(* Logix 5000 project; controller cal1632 1756-L62 rev 16.20; software revision 16.05; part 53 of 57 *)
(* tags used below, declared in another part *)
   AFI : BOOL;
   FAULT : BOOL;
   p01_recipe_active : recipe;
   p01r02_plc_scan_time_in_sec : REAL;
   p01r09_pb_global_reset : BOOL;
   p01r09_request_line_jog : BOOL;
   p01r13_line_running : BOOL;
   p01r13_line_slow_ramp : BOOL;
   p01r13_permissive_drives : BOOL;
   p02_real_from_hmi : hmi_real;
   p25_ao_selected_speed : REAL;
   p25r09_mode_thread : BOOL;
   p25r09_pb_jog_fwd : BOOL;
   p25r09_pb_jog_rev : BOOL;
   p29_ai_wa_torque : REAL;
   p29_ai_wb_torque : REAL;
   p29_ai_wdr_lc : REAL;
   p29_ao_wdra_selected_speed : REAL;
   p29_ao_wdrb_selected_speed : REAL;
   p29_di_wa_brake : BOOL;
   p29_di_wa_motor : BOOL;
   p29_di_wdr_a_start : BOOL;
   p29_di_wdr_a_stop : BOOL;
   p29_di_wdr_b_start : BOOL;
   p29_di_wdr_b_stop : BOOL;
   p29_di_wdr_index_fwd : BOOL;
   p29_di_wdr_jog : BOOL;
   p29_param_soak : REAL;
   p29_param_winder_jog_speed : REAL;
   p29_wda_control_word : INT;
   p29_wda_status_word : INT;
   p29_wda_vfd : ABB_PROTOCOL_VFD;
   p29_wdb_control_word : INT;
   p29_wdb_status_word : INT;
   p29_wdb_vfd : ABB_PROTOCOL_VFD;
   p29r02_tension_dev_max : REAL;
   p29r02_tension_dev_min : REAL;
   p29r02_wa_calc_torque_ref : REAL;
   p29r02_wb_calc_torque_ref : REAL;
   p29r09_torque_mode : BOOL;
   p29r09_winder_a_active : BOOL;
   p29r09_winder_b_active : BOOL;
   p29r10_index_active : BOOL;
   p29r10_speed_offset : REAL;
   p29r11_index_active : BOOL;
   p29r11_speed_offset : REAL;
   p29r15 : routine;
   p29r15_accel_rate : REAL;
   p29r15_ao_torque : REAL;
   p29r15_const_torque_ref : REAL;
   p29r15_decel_rate : REAL;
   p29r15_fast_accel_rate : REAL;
   p29r15_fast_decel_rate : REAL;
   p29r15_index_start_torque : REAL;
   p29r15_jog_torque_ref : REAL;
   p29r15_request_jog_fwd : BOOL;
   p29r15_request_run : BOOL;
   p29r15_request_thread_fwd : BOOL;
   p29r15_request_thread_rev : BOOL;
   p29r15_run_permissive : BOOL;
   p29r15_selected_speed : REAL;
   p29r15_selected_torque : REAL;
   p29r15_soak_active : BOOL;
   p29r15_state : DINT;
   p29r15_tension_ok : BOOL;
   p29r15_thread_torque_ref : REAL;
   p29r15_timer_fault : TIMER[10];
   p29r15_timer_warning : TIMER[4];
   p29r15_torque_acc_rate : REAL;
   p29r15_torque_boost_acc_rate : REAL;
   p29r15_torque_boost_dec_rate : REAL;
   p29r15_torque_boost_ref : REAL;
   p29r15_torque_boost_timer : TIMER;
   p29r15_torque_dec_rate : REAL;
   p29r15_torque_fast_acc_rate : REAL;
   p29r15_torque_fast_dec_rate : REAL;
   p29r15_torque_high_ref : REAL;
   p29r15_torque_low_ref : REAL;
   p29r15_torque_mode_acc_rate : REAL;
   p29r15_torque_mode_dec_rate : REAL;
   p29r15_torque_ramp : SYS_ACC_DEC_RAMP;
   p29r15_torque_soak_acc_rate : REAL;
   p29r15_torque_soak_dec_rate : REAL;
   p29r15_torque_start_timer : TIMER;
   p29r15_wda_vfd_start_request : BOOL;
   p29r15_wdra_accel_decel : SYS_ACC_DEC_RAMP;
   p29r15_wdra_active : BOOL;
   p29r15_wdra_ramped_speed : REAL;
   p29r15_zero_speed : BOOL;
   p29r16 : routine;
   p29r16_accel_rate : REAL;
   p29r16_ao_torque : REAL;
   p29r16_const_torque_ref : REAL;
   p29r16_decel_rate : REAL;
   p29r16_fast_accel_rate : REAL;
   p29r16_fast_decel_rate : REAL;
   p29r16_index_start_torque : REAL;
   p29r16_jog_torque_ref : REAL;
   p29r16_request_jog_fwd : BOOL;
   p29r16_request_run : BOOL;
   p29r16_request_thread_fwd : BOOL;
   p29r16_request_thread_rev : BOOL;
   p29r16_run_permissive : BOOL;
   p29r16_selected_speed : REAL;
   p29r16_selected_torque : REAL;
   p29r16_soak_active : BOOL;
   p29r16_state : DINT;
   p29r16_tension_ok : BOOL;
   p29r16_thread_torque_ref : REAL;
   p29r16_timer_fault : TIMER[10];
   p29r16_torque_acc_rate : REAL;
   p29r16_torque_boost_acc_rate : REAL;
   p29r16_torque_boost_dec_rate : REAL;
   p29r16_torque_boost_ref : REAL;
   p29r16_torque_boost_timer : TIMER;
   p29r16_torque_dec_rate : REAL;
   p29r16_torque_fast_acc_rate : REAL;
   p29r16_torque_fast_dec_rate : REAL;
   p29r16_torque_high_ref : REAL;
   p29r16_torque_low_ref : REAL;
   p29r16_torque_mode_acc_rate : REAL;
   p29r16_torque_mode_dec_rate : REAL;
   p29r16_torque_ramp : SYS_ACC_DEC_RAMP;
   p29r16_torque_soak_acc_rate : REAL;
   p29r16_torque_soak_dec_rate : REAL;
   p29r16_torque_start_timer : TIMER;
   p29r16_vfd_start_request : BOOL;
   p29r16_wdrb_accel_decel : SYS_ACC_DEC_RAMP;
   p29r16_wdrb_active : BOOL;
   p29r16_wdrb_ramped_speed : REAL;
   p29r16_zero_speed : BOOL;
(* P29_Winder, continued *)

ROUTINE R15_Winder_A_VFD   (* ladder *)
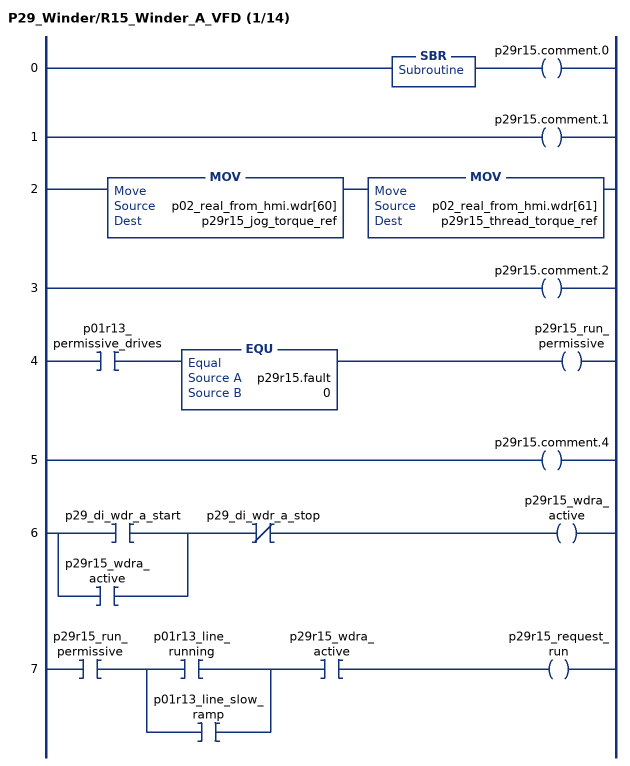
   0: SBR()OTE(p29r15.comment.0);
   1: OTE(p29r15.comment.1);
   2: MOV(p02_real_from_hmi.wdr[60],p29r15_jog_torque_ref)MOV(p02_real_from_hmi.wdr[61],p29r15_thread_torque_ref);
   3: OTE(p29r15.comment.2);
   4: XIC(p01r13_permissive_drives)EQU(p29r15.fault,0)OTE(p29r15_run_permissive);
   5: OTE(p29r15.comment.4);
   6: [XIC(p29_di_wdr_a_start) ,XIC(p29r15_wdra_active) ]XIO(p29_di_wdr_a_stop)OTE(p29r15_wdra_active);
   7: XIC(p29r15_run_permissive)[XIC(p01r13_line_running) ,XIC(p01r13_line_slow_ramp) ]XIC(p29r15_wdra_active)OTE(p29r15_request_run);
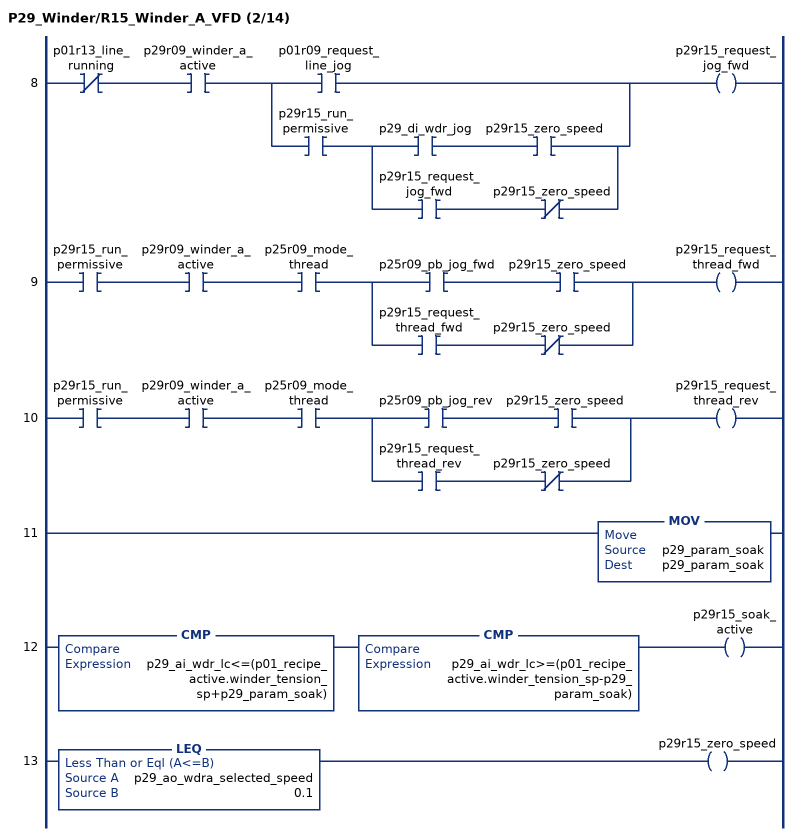
   8: XIO(p01r13_line_running)XIC(p29r09_winder_a_active)[XIC(p01r09_request_line_jog) ,XIC(p29r15_run_permissive) [XIC(p29_di_wdr_jog) XIC(p29r15_zero_speed) ,XIC(p29r15_request_jog_fwd) XIO(p29r15_zero_speed) ] ]OTE(p29r15_request_jog_fwd);
   9: XIC(p29r15_run_permissive)XIC(p29r09_winder_a_active)XIC(p25r09_mode_thread)[XIC(p25r09_pb_jog_fwd) XIC(p29r15_zero_speed) ,XIC(p29r15_request_thread_fwd) XIO(p29r15_zero_speed) ]OTE(p29r15_request_thread_fwd);
   10: XIC(p29r15_run_permissive)XIC(p29r09_winder_a_active)XIC(p25r09_mode_thread)[XIC(p25r09_pb_jog_rev) XIC(p29r15_zero_speed) ,XIC(p29r15_request_thread_rev) XIO(p29r15_zero_speed) ]OTE(p29r15_request_thread_rev);
   11: MOV(p29_param_soak,p29_param_soak);
   12: CMP(p29_ai_wdr_lc<=(p01_recipe_active.winder_tension_sp+p29_param_soak))CMP(p29_ai_wdr_lc>=(p01_recipe_active.winder_tension_sp-p29_param_soak))OTE(p29r15_soak_active);
   13: LEQ(p29_ao_wdra_selected_speed,0.1)OTE(p29r15_zero_speed);
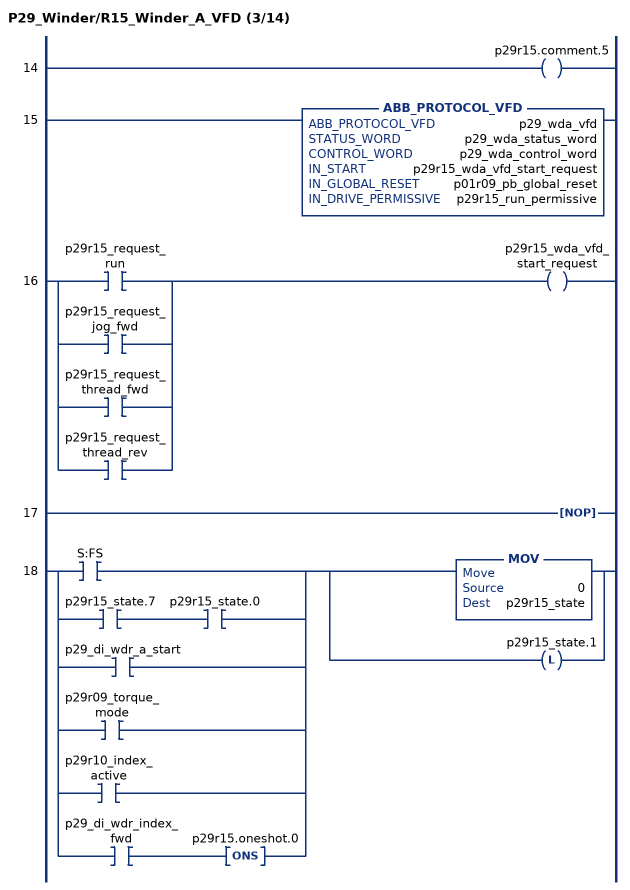
   14: OTE(p29r15.comment.5);
   15: ABB_PROTOCOL_VFD(p29_wda_vfd,p29_wda_status_word,p29_wda_control_word,p29r15_wda_vfd_start_request,p01r09_pb_global_reset,p29r15_run_permissive);
   16: [XIC(p29r15_request_run) ,XIC(p29r15_request_jog_fwd) ,XIC(p29r15_request_thread_fwd) ,XIC(p29r15_request_thread_rev) ]OTE(p29r15_wda_vfd_start_request);
   17: NOP();
   18: [XIC(S:FS) ,XIC(p29r15_state.7) XIC(p29r15_state.0) ,XIC(p29_di_wdr_a_start) ,XIC(p29r09_torque_mode) ,XIC(p29r10_index_active) ,XIC(p29_di_wdr_index_fwd) ONS(p29r15.oneshot.0) ][MOV(0,p29r15_state) ,OTL(p29r15_state.1) ];
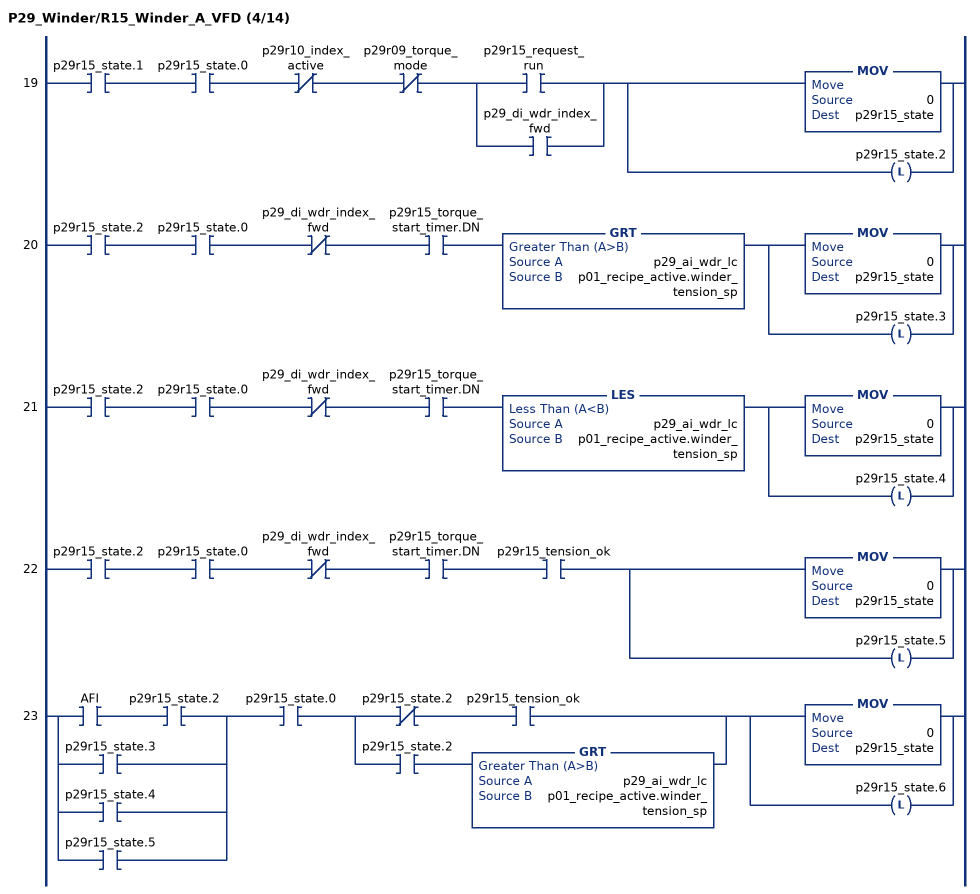
   19: XIC(p29r15_state.1)XIC(p29r15_state.0)XIO(p29r10_index_active)XIO(p29r09_torque_mode)[XIC(p29r15_request_run) ,XIC(p29_di_wdr_index_fwd) ][MOV(0,p29r15_state) ,OTL(p29r15_state.2) ];
   20: XIC(p29r15_state.2)XIC(p29r15_state.0)XIO(p29_di_wdr_index_fwd)XIC(p29r15_torque_start_timer.DN)GRT(p29_ai_wdr_lc,p01_recipe_active.winder_tension_sp)[MOV(0,p29r15_state) ,OTL(p29r15_state.3) ];
   21: XIC(p29r15_state.2)XIC(p29r15_state.0)XIO(p29_di_wdr_index_fwd)XIC(p29r15_torque_start_timer.DN)LES(p29_ai_wdr_lc,p01_recipe_active.winder_tension_sp)[MOV(0,p29r15_state) ,OTL(p29r15_state.4) ];
   22: XIC(p29r15_state.2)XIC(p29r15_state.0)XIO(p29_di_wdr_index_fwd)XIC(p29r15_torque_start_timer.DN)XIC(p29r15_tension_ok)[MOV(0,p29r15_state) ,OTL(p29r15_state.5) ];
   23: [XIC(AFI) XIC(p29r15_state.2) ,XIC(p29r15_state.3) ,XIC(p29r15_state.4) ,XIC(p29r15_state.5) ]XIC(p29r15_state.0)[XIO(p29r15_state.2) XIC(p29r15_tension_ok) ,XIC(p29r15_state.2) GRT(p29_ai_wdr_lc,p01_recipe_active.winder_tension_sp) ][MOV(0,p29r15_state) ,OTL(p29r15_state.6) ];
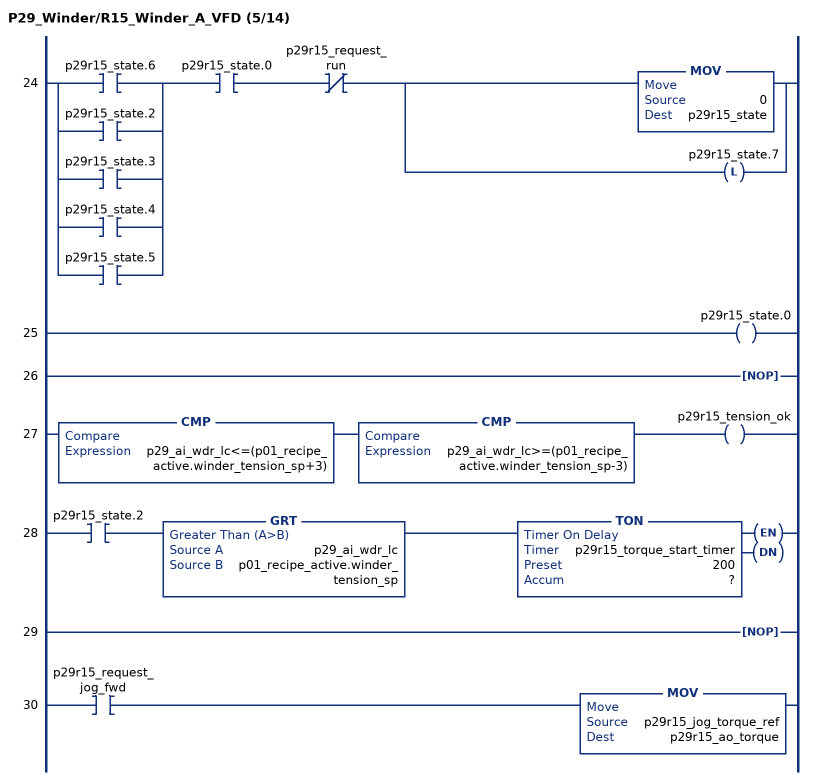
   24: [XIC(p29r15_state.6) ,XIC(p29r15_state.2) ,XIC(p29r15_state.3) ,XIC(p29r15_state.4) ,XIC(p29r15_state.5) ]XIC(p29r15_state.0)XIO(p29r15_request_run)[MOV(0,p29r15_state) ,OTL(p29r15_state.7) ];
   25: OTE(p29r15_state.0);
   26: NOP();
   27: CMP(p29_ai_wdr_lc<=(p01_recipe_active.winder_tension_sp+3))CMP(p29_ai_wdr_lc>=(p01_recipe_active.winder_tension_sp-3))OTE(p29r15_tension_ok);
   28: XIC(p29r15_state.2)GRT(p29_ai_wdr_lc,p01_recipe_active.winder_tension_sp)TON(p29r15_torque_start_timer,?,?);
   29: NOP();
   30: XIC(p29r15_request_jog_fwd)MOV(p29r15_jog_torque_ref,p29r15_ao_torque);
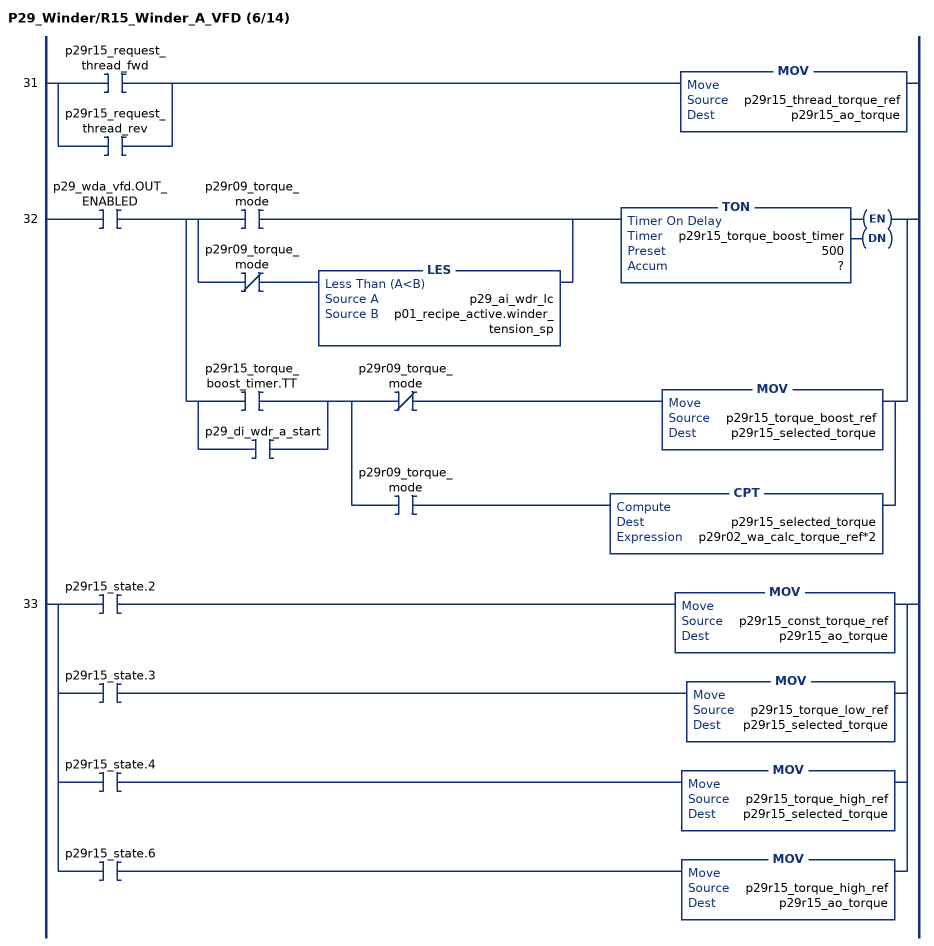
   31: [XIC(p29r15_request_thread_fwd) ,XIC(p29r15_request_thread_rev) ]MOV(p29r15_thread_torque_ref,p29r15_ao_torque);
   32: XIC(p29_wda_vfd.OUT_ENABLED)[[XIC(p29r09_torque_mode) ,XIO(p29r09_torque_mode) LES(p29_ai_wdr_lc,p01_recipe_active.winder_tension_sp) ] TON(p29r15_torque_boost_timer,?,?) ,[XIC(p29r15_torque_boost_timer.TT) ,XIC(p29_di_wdr_a_start) ] [XIO(p29r09_torque_mode) MOV(p29r15_torque_boost_ref,p29r15_selected_torque) ,XIC(p29r09_torque_mode) CPT(p29r15_selected_torque,p29r02_wa_calc_torque_ref*2) ] ];
   33: [XIC(p29r15_state.2) MOV(p29r15_const_torque_ref,p29r15_ao_torque) ,XIC(p29r15_state.3) MOV(p29r15_torque_low_ref,p29r15_selected_torque) ,XIC(p29r15_state.4) MOV(p29r15_torque_high_ref,p29r15_selected_torque) ,XIC(p29r15_state.6) MOV(p29r15_torque_high_ref,p29r15_ao_torque) ];
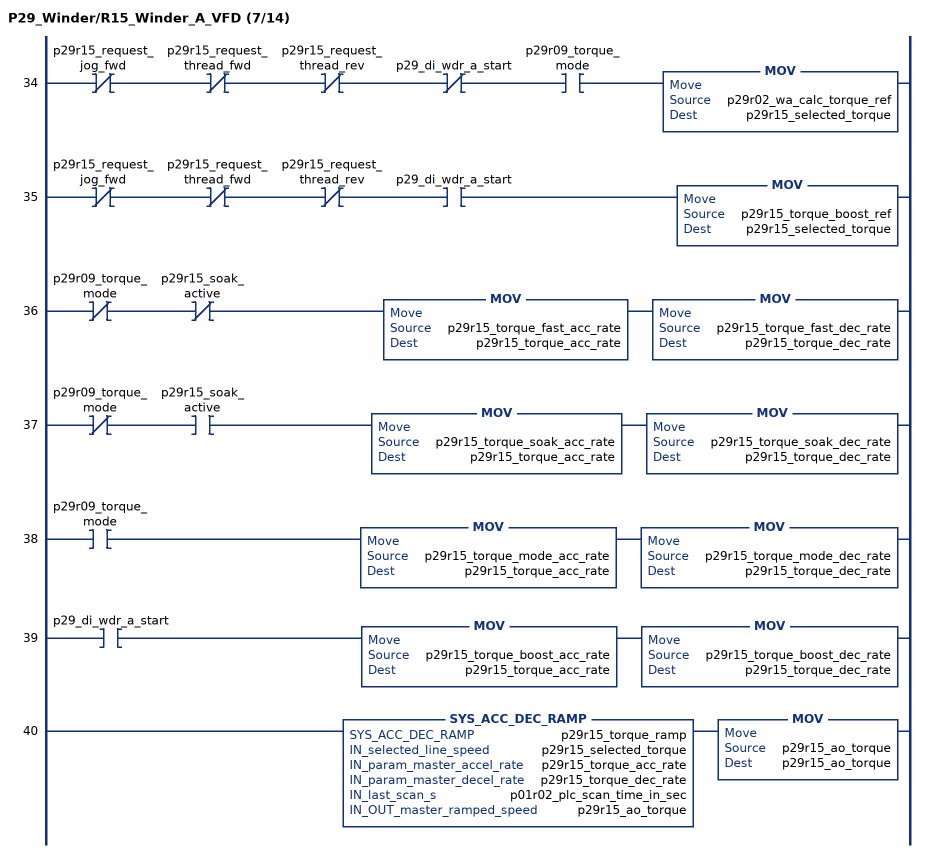
   34: XIO(p29r15_request_jog_fwd)XIO(p29r15_request_thread_fwd)XIO(p29r15_request_thread_rev)XIO(p29_di_wdr_a_start)XIC(p29r09_torque_mode)MOV(p29r02_wa_calc_torque_ref,p29r15_selected_torque);
   35: XIO(p29r15_request_jog_fwd)XIO(p29r15_request_thread_fwd)XIO(p29r15_request_thread_rev)XIC(p29_di_wdr_a_start)MOV(p29r15_torque_boost_ref,p29r15_selected_torque);
   36: XIO(p29r09_torque_mode)XIO(p29r15_soak_active)MOV(p29r15_torque_fast_acc_rate,p29r15_torque_acc_rate)MOV(p29r15_torque_fast_dec_rate,p29r15_torque_dec_rate);
   37: XIO(p29r09_torque_mode)XIC(p29r15_soak_active)MOV(p29r15_torque_soak_acc_rate,p29r15_torque_acc_rate)MOV(p29r15_torque_soak_dec_rate,p29r15_torque_dec_rate);
   38: XIC(p29r09_torque_mode)MOV(p29r15_torque_mode_acc_rate,p29r15_torque_acc_rate)MOV(p29r15_torque_mode_dec_rate,p29r15_torque_dec_rate);
   39: XIC(p29_di_wdr_a_start)MOV(p29r15_torque_boost_acc_rate,p29r15_torque_acc_rate)MOV(p29r15_torque_boost_dec_rate,p29r15_torque_dec_rate);
   40: SYS_ACC_DEC_RAMP(p29r15_torque_ramp,p29r15_selected_torque,p29r15_torque_acc_rate,p29r15_torque_dec_rate,p01r02_plc_scan_time_in_sec,p29r15_ao_torque)MOV(p29r15_ao_torque,p29r15_ao_torque);
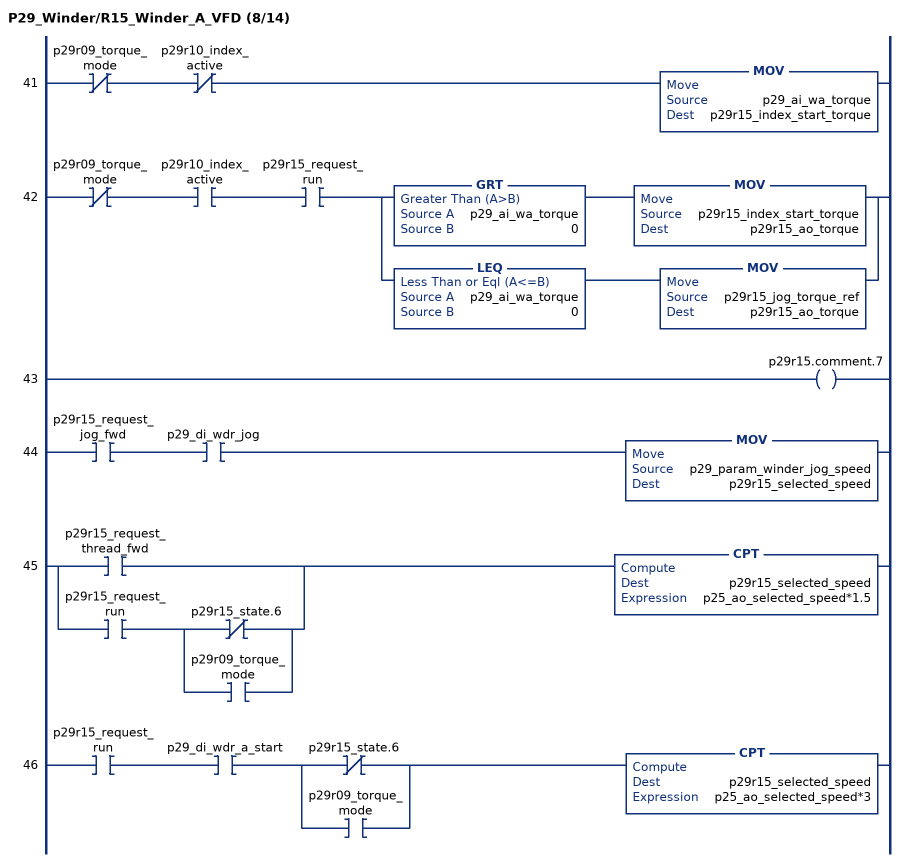
   41: XIO(p29r09_torque_mode)XIO(p29r10_index_active)MOV(p29_ai_wa_torque,p29r15_index_start_torque);
   42: XIO(p29r09_torque_mode)XIC(p29r10_index_active)XIC(p29r15_request_run)[GRT(p29_ai_wa_torque,0) MOV(p29r15_index_start_torque,p29r15_ao_torque) ,LEQ(p29_ai_wa_torque,0) MOV(p29r15_jog_torque_ref,p29r15_ao_torque) ];
   43: OTE(p29r15.comment.7);
   44: XIC(p29r15_request_jog_fwd)XIC(p29_di_wdr_jog)MOV(p29_param_winder_jog_speed,p29r15_selected_speed);
   45: [XIC(p29r15_request_thread_fwd) ,XIC(p29r15_request_run) [XIO(p29r15_state.6) ,XIC(p29r09_torque_mode) ] ]CPT(p29r15_selected_speed,p25_ao_selected_speed*1.5);
   46: XIC(p29r15_request_run)XIC(p29_di_wdr_a_start)[XIO(p29r15_state.6) ,XIC(p29r09_torque_mode) ]CPT(p29r15_selected_speed,p25_ao_selected_speed*3);
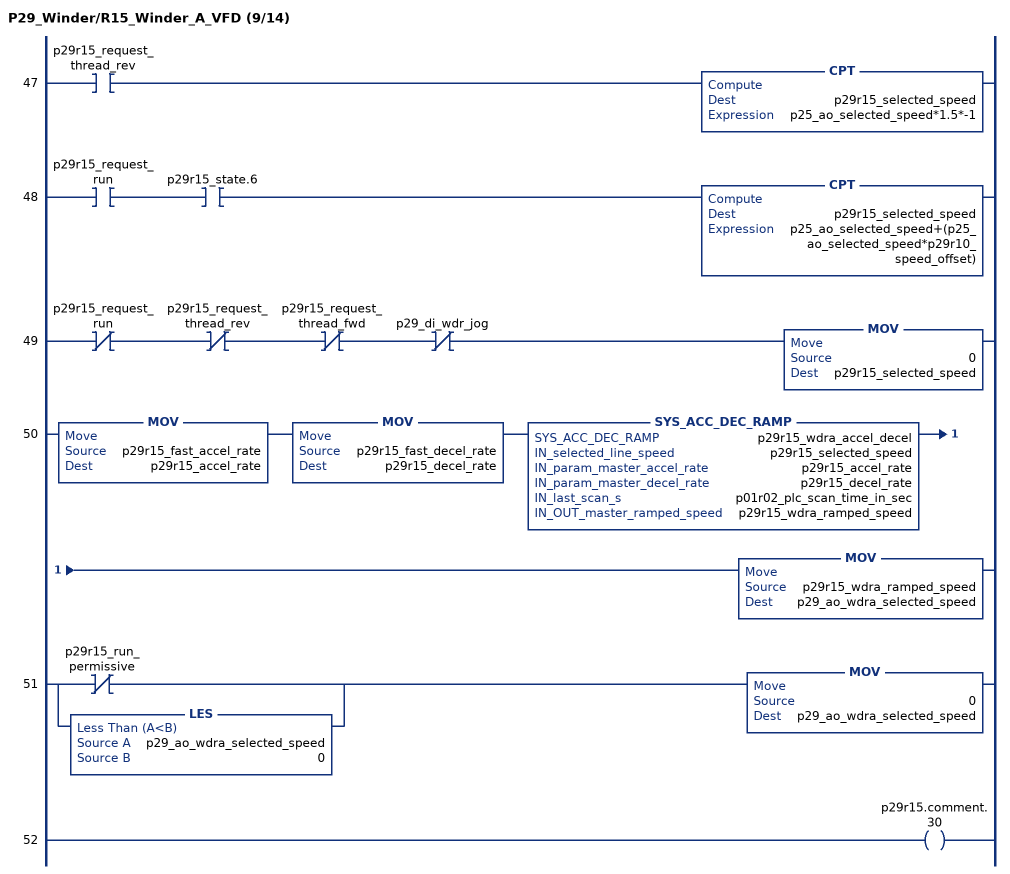
   47: XIC(p29r15_request_thread_rev)CPT(p29r15_selected_speed,p25_ao_selected_speed*1.5*-1);
   48: XIC(p29r15_request_run)XIC(p29r15_state.6)CPT(p29r15_selected_speed,p25_ao_selected_speed+(p25_ao_selected_speed*p29r10_speed_offset));
   49: XIO(p29r15_request_run)XIO(p29r15_request_thread_rev)XIO(p29r15_request_thread_fwd)XIO(p29_di_wdr_jog)MOV(0,p29r15_selected_speed);
   50: MOV(p29r15_fast_accel_rate,p29r15_accel_rate)MOV(p29r15_fast_decel_rate,p29r15_decel_rate)SYS_ACC_DEC_RAMP(p29r15_wdra_accel_decel,p29r15_selected_speed,p29r15_accel_rate,p29r15_decel_rate,p01r02_plc_scan_time_in_sec,p29r15_wdra_ramped_speed)MOV(p29r15_wdra_ramped_speed,p29_ao_wdra_selected_speed);
   51: [XIO(p29r15_run_permissive) ,LES(p29_ao_wdra_selected_speed,0) ]MOV(0,p29_ao_wdra_selected_speed);
   52: OTE(p29r15.comment.30);
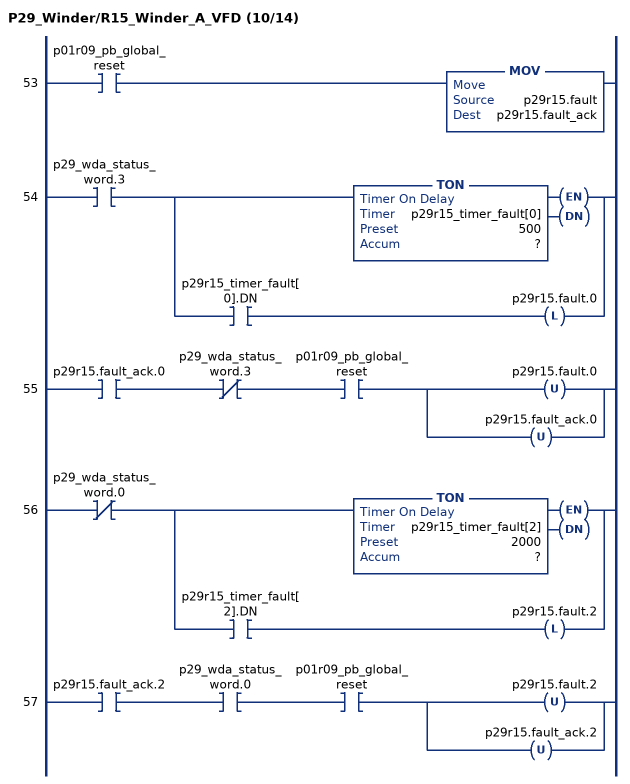
   53: XIC(p01r09_pb_global_reset)MOV(p29r15.fault,p29r15.fault_ack);
   54: XIC(p29_wda_status_word.3)[TON(p29r15_timer_fault[0],?,?) ,XIC(p29r15_timer_fault[0].DN) OTL(p29r15.fault.0) ];
   55: XIC(p29r15.fault_ack.0)XIO(p29_wda_status_word.3)XIC(p01r09_pb_global_reset)[OTU(p29r15.fault.0) ,OTU(p29r15.fault_ack.0) ];
   56: XIO(p29_wda_status_word.0)[TON(p29r15_timer_fault[2],?,?) ,XIC(p29r15_timer_fault[2].DN) OTL(p29r15.fault.2) ];
   57: XIC(p29r15.fault_ack.2)XIC(p29_wda_status_word.0)XIC(p01r09_pb_global_reset)[OTU(p29r15.fault.2) ,OTU(p29r15.fault_ack.2) ];
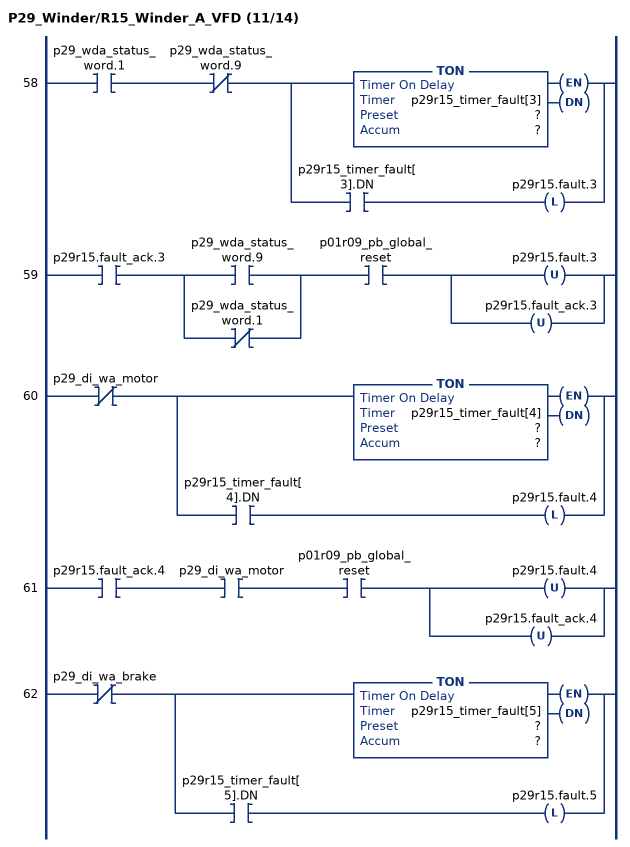
   58: XIC(p29_wda_status_word.1)XIO(p29_wda_status_word.9)[TON(p29r15_timer_fault[3],?,?) ,XIC(p29r15_timer_fault[3].DN) OTL(p29r15.fault.3) ];
   59: XIC(p29r15.fault_ack.3)[XIC(p29_wda_status_word.9) ,XIO(p29_wda_status_word.1) ]XIC(p01r09_pb_global_reset)[OTU(p29r15.fault.3) ,OTU(p29r15.fault_ack.3) ];
   60: XIO(p29_di_wa_motor)[TON(p29r15_timer_fault[4],?,?) ,XIC(p29r15_timer_fault[4].DN) OTL(p29r15.fault.4) ];
   61: XIC(p29r15.fault_ack.4)XIC(p29_di_wa_motor)XIC(p01r09_pb_global_reset)[OTU(p29r15.fault.4) ,OTU(p29r15.fault_ack.4) ];
   62: XIO(p29_di_wa_brake)[TON(p29r15_timer_fault[5],?,?) ,XIC(p29r15_timer_fault[5].DN) OTL(p29r15.fault.5) ];
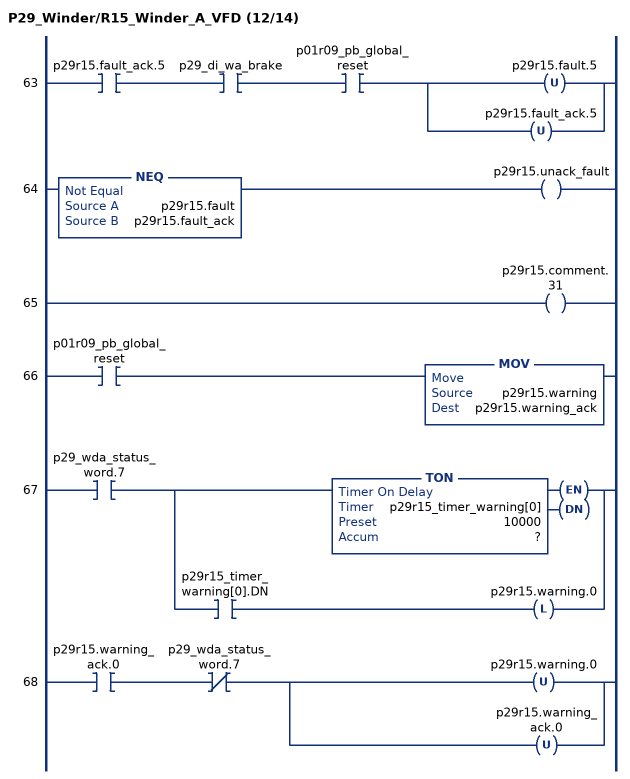
   63: XIC(p29r15.fault_ack.5)XIC(p29_di_wa_brake)XIC(p01r09_pb_global_reset)[OTU(p29r15.fault.5) ,OTU(p29r15.fault_ack.5) ];
   64: NEQ(p29r15.fault,p29r15.fault_ack)OTE(p29r15.unack_fault);
   65: OTE(p29r15.comment.31);
   66: XIC(p01r09_pb_global_reset)MOV(p29r15.warning,p29r15.warning_ack);
   67: XIC(p29_wda_status_word.7)[TON(p29r15_timer_warning[0],?,?) ,XIC(p29r15_timer_warning[0].DN) OTL(p29r15.warning.0) ];
   68: XIC(p29r15.warning_ack.0)XIO(p29_wda_status_word.7)[OTU(p29r15.warning.0) ,OTU(p29r15.warning_ack.0) ];
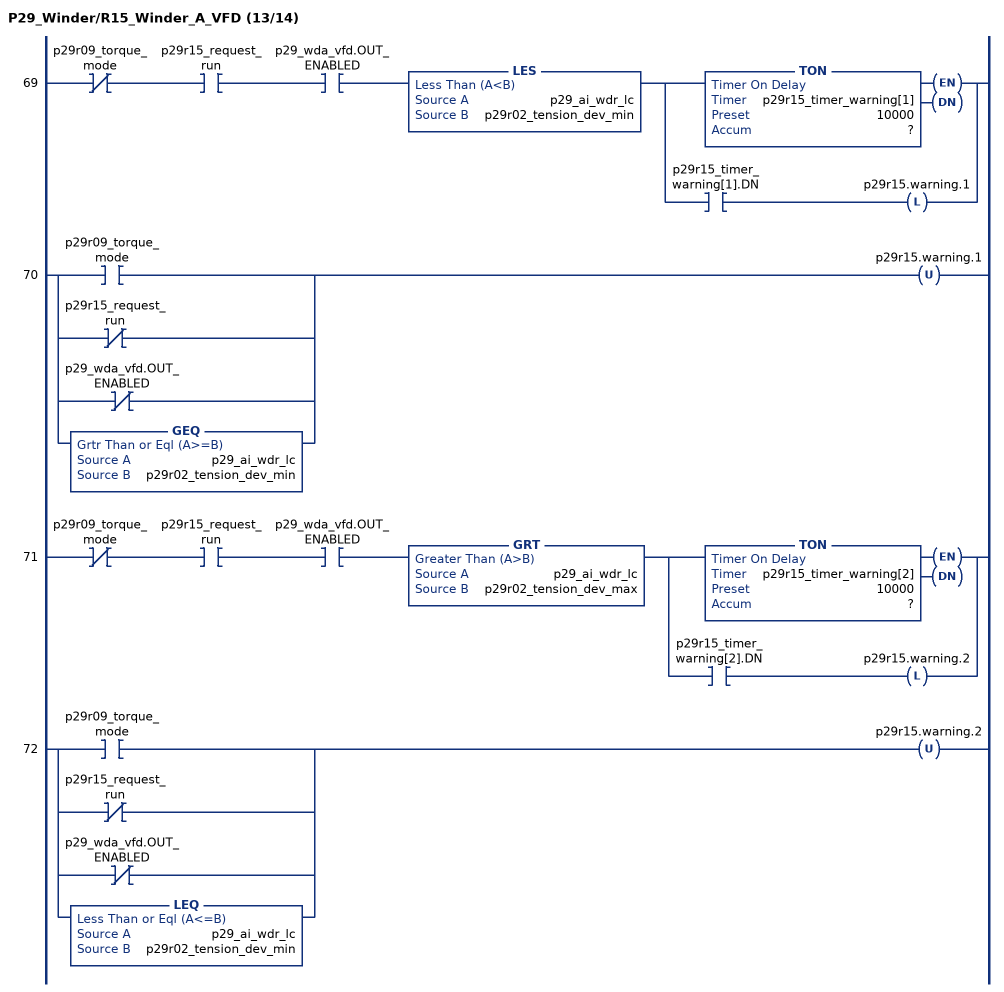
   69: XIO(p29r09_torque_mode)XIC(p29r15_request_run)XIC(p29_wda_vfd.OUT_ENABLED)LES(p29_ai_wdr_lc,p29r02_tension_dev_min)[TON(p29r15_timer_warning[1],?,?) ,XIC(p29r15_timer_warning[1].DN) OTL(p29r15.warning.1) ];
   70: [XIC(p29r09_torque_mode) ,XIO(p29r15_request_run) ,XIO(p29_wda_vfd.OUT_ENABLED) ,GEQ(p29_ai_wdr_lc,p29r02_tension_dev_min) ]OTU(p29r15.warning.1);
   71: XIO(p29r09_torque_mode)XIC(p29r15_request_run)XIC(p29_wda_vfd.OUT_ENABLED)GRT(p29_ai_wdr_lc,p29r02_tension_dev_max)[TON(p29r15_timer_warning[2],?,?) ,XIC(p29r15_timer_warning[2].DN) OTL(p29r15.warning.2) ];
   72: [XIC(p29r09_torque_mode) ,XIO(p29r15_request_run) ,XIO(p29_wda_vfd.OUT_ENABLED) ,LEQ(p29_ai_wdr_lc,p29r02_tension_dev_min) ]OTU(p29r15.warning.2);
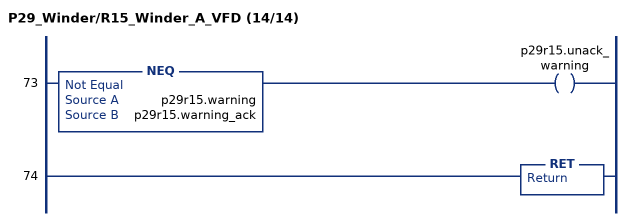
   73: NEQ(p29r15.warning,p29r15.warning_ack)OTE(p29r15.unack_warning);
   74: RET();
END_ROUTINE

ROUTINE R16_Winder_B_VFD   (* ladder *)
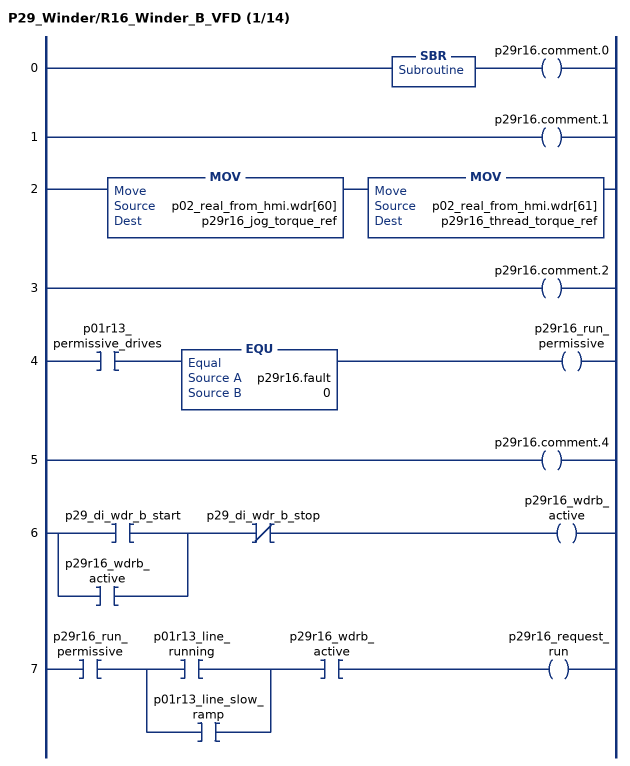
   0: SBR()OTE(p29r16.comment.0);
   1: OTE(p29r16.comment.1);
   2: MOV(p02_real_from_hmi.wdr[60],p29r16_jog_torque_ref)MOV(p02_real_from_hmi.wdr[61],p29r16_thread_torque_ref);
   3: OTE(p29r16.comment.2);
   4: XIC(p01r13_permissive_drives)EQU(p29r16.fault,0)OTE(p29r16_run_permissive);
   5: OTE(p29r16.comment.4);
   6: [XIC(p29_di_wdr_b_start) ,XIC(p29r16_wdrb_active) ]XIO(p29_di_wdr_b_stop)OTE(p29r16_wdrb_active);
   7: XIC(p29r16_run_permissive)[XIC(p01r13_line_running) ,XIC(p01r13_line_slow_ramp) ]XIC(p29r16_wdrb_active)OTE(p29r16_request_run);
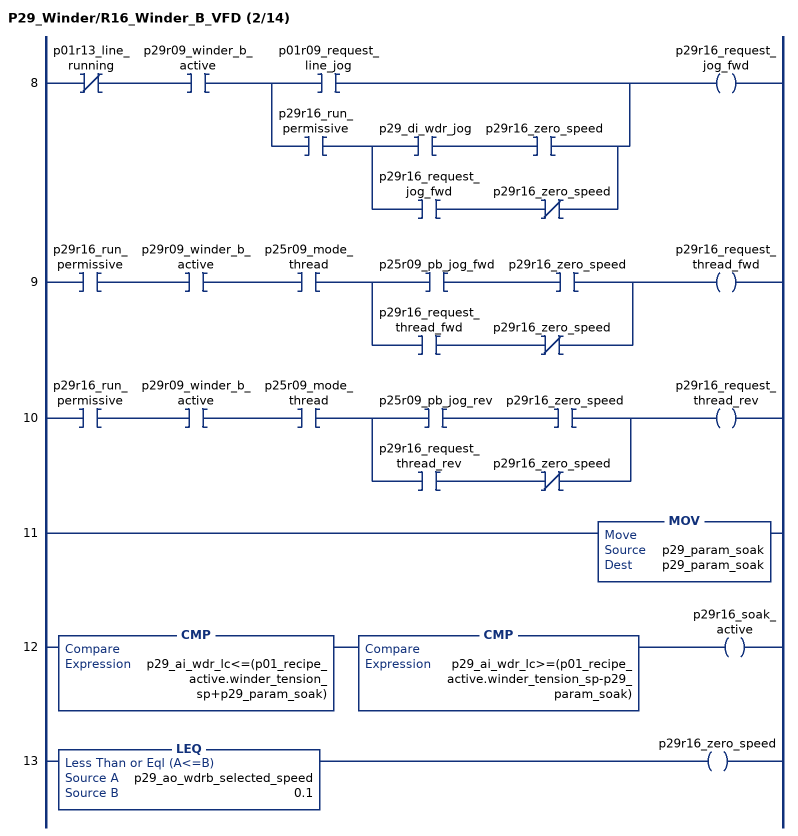
   8: XIO(p01r13_line_running)XIC(p29r09_winder_b_active)[XIC(p01r09_request_line_jog) ,XIC(p29r16_run_permissive) [XIC(p29_di_wdr_jog) XIC(p29r16_zero_speed) ,XIC(p29r16_request_jog_fwd) XIO(p29r16_zero_speed) ] ]OTE(p29r16_request_jog_fwd);
   9: XIC(p29r16_run_permissive)XIC(p29r09_winder_b_active)XIC(p25r09_mode_thread)[XIC(p25r09_pb_jog_fwd) XIC(p29r16_zero_speed) ,XIC(p29r16_request_thread_fwd) XIO(p29r16_zero_speed) ]OTE(p29r16_request_thread_fwd);
   10: XIC(p29r16_run_permissive)XIC(p29r09_winder_b_active)XIC(p25r09_mode_thread)[XIC(p25r09_pb_jog_rev) XIC(p29r16_zero_speed) ,XIC(p29r16_request_thread_rev) XIO(p29r16_zero_speed) ]OTE(p29r16_request_thread_rev);
   11: MOV(p29_param_soak,p29_param_soak);
   12: CMP(p29_ai_wdr_lc<=(p01_recipe_active.winder_tension_sp+p29_param_soak))CMP(p29_ai_wdr_lc>=(p01_recipe_active.winder_tension_sp-p29_param_soak))OTE(p29r16_soak_active);
   13: LEQ(p29_ao_wdrb_selected_speed,0.1)OTE(p29r16_zero_speed);
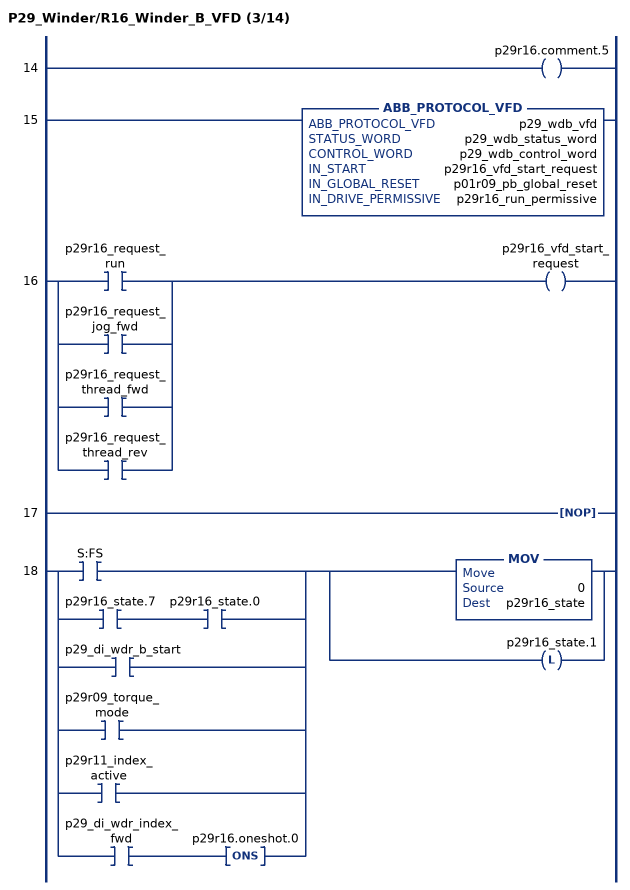
   14: OTE(p29r16.comment.5);
   15: ABB_PROTOCOL_VFD(p29_wdb_vfd,p29_wdb_status_word,p29_wdb_control_word,p29r16_vfd_start_request,p01r09_pb_global_reset,p29r16_run_permissive);
   16: [XIC(p29r16_request_run) ,XIC(p29r16_request_jog_fwd) ,XIC(p29r16_request_thread_fwd) ,XIC(p29r16_request_thread_rev) ]OTE(p29r16_vfd_start_request);
   17: NOP();
   18: [XIC(S:FS) ,XIC(p29r16_state.7) XIC(p29r16_state.0) ,XIC(p29_di_wdr_b_start) ,XIC(p29r09_torque_mode) ,XIC(p29r11_index_active) ,XIC(p29_di_wdr_index_fwd) ONS(p29r16.oneshot.0) ][MOV(0,p29r16_state) ,OTL(p29r16_state.1) ];
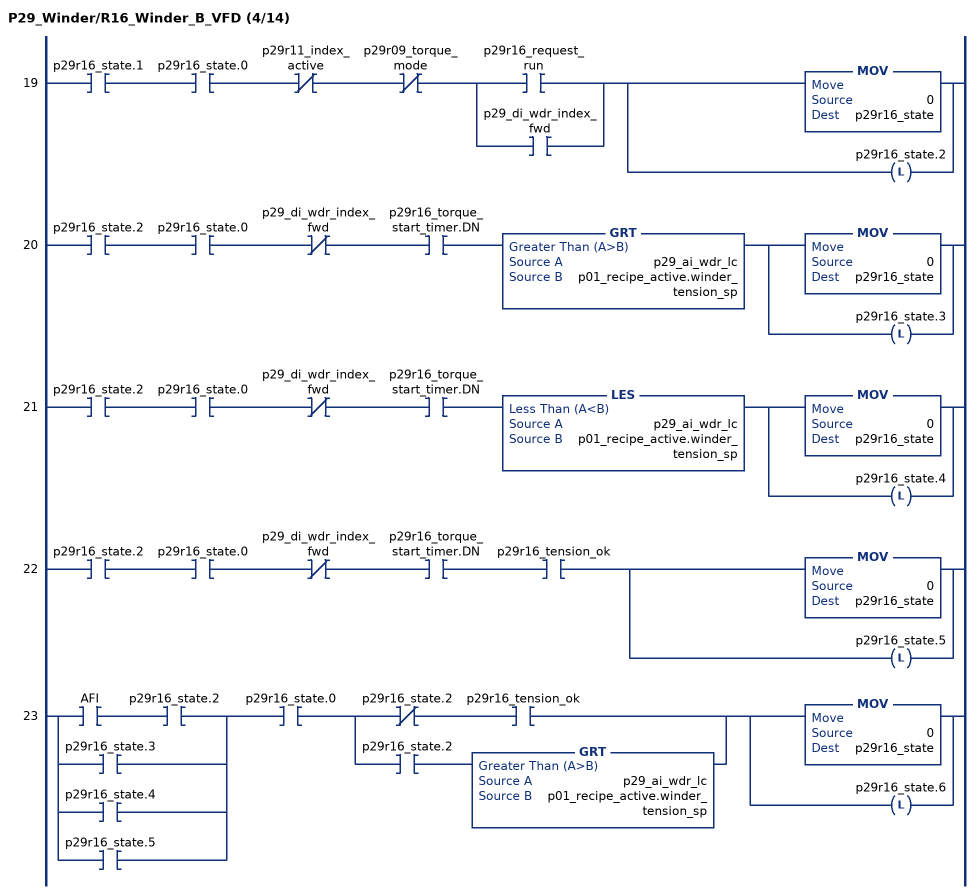
   19: XIC(p29r16_state.1)XIC(p29r16_state.0)XIO(p29r11_index_active)XIO(p29r09_torque_mode)[XIC(p29r16_request_run) ,XIC(p29_di_wdr_index_fwd) ][MOV(0,p29r16_state) ,OTL(p29r16_state.2) ];
   20: XIC(p29r16_state.2)XIC(p29r16_state.0)XIO(p29_di_wdr_index_fwd)XIC(p29r16_torque_start_timer.DN)GRT(p29_ai_wdr_lc,p01_recipe_active.winder_tension_sp)[MOV(0,p29r16_state) ,OTL(p29r16_state.3) ];
   21: XIC(p29r16_state.2)XIC(p29r16_state.0)XIO(p29_di_wdr_index_fwd)XIC(p29r16_torque_start_timer.DN)LES(p29_ai_wdr_lc,p01_recipe_active.winder_tension_sp)[MOV(0,p29r16_state) ,OTL(p29r16_state.4) ];
   22: XIC(p29r16_state.2)XIC(p29r16_state.0)XIO(p29_di_wdr_index_fwd)XIC(p29r16_torque_start_timer.DN)XIC(p29r16_tension_ok)[MOV(0,p29r16_state) ,OTL(p29r16_state.5) ];
   23: [XIC(AFI) XIC(p29r16_state.2) ,XIC(p29r16_state.3) ,XIC(p29r16_state.4) ,XIC(p29r16_state.5) ]XIC(p29r16_state.0)[XIO(p29r16_state.2) XIC(p29r16_tension_ok) ,XIC(p29r16_state.2) GRT(p29_ai_wdr_lc,p01_recipe_active.winder_tension_sp) ][MOV(0,p29r16_state) ,OTL(p29r16_state.6) ];
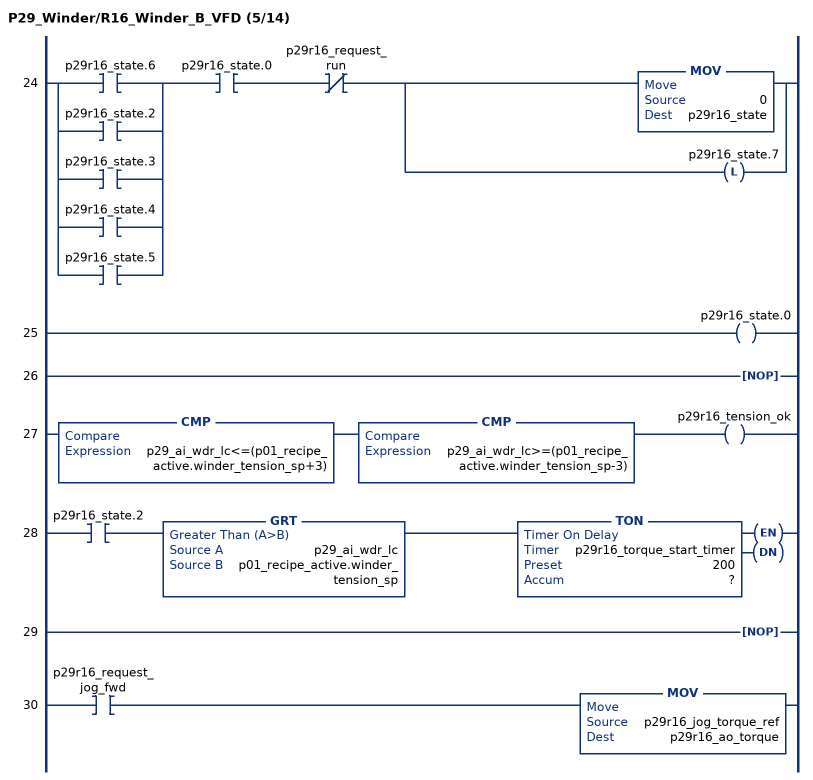
   24: [XIC(p29r16_state.6) ,XIC(p29r16_state.2) ,XIC(p29r16_state.3) ,XIC(p29r16_state.4) ,XIC(p29r16_state.5) ]XIC(p29r16_state.0)XIO(p29r16_request_run)[MOV(0,p29r16_state) ,OTL(p29r16_state.7) ];
   25: OTE(p29r16_state.0);
   26: NOP();
   27: CMP(p29_ai_wdr_lc<=(p01_recipe_active.winder_tension_sp+3))CMP(p29_ai_wdr_lc>=(p01_recipe_active.winder_tension_sp-3))OTE(p29r16_tension_ok);
   28: XIC(p29r16_state.2)GRT(p29_ai_wdr_lc,p01_recipe_active.winder_tension_sp)TON(p29r16_torque_start_timer,?,?);
   29: NOP();
   30: XIC(p29r16_request_jog_fwd)MOV(p29r16_jog_torque_ref,p29r16_ao_torque);
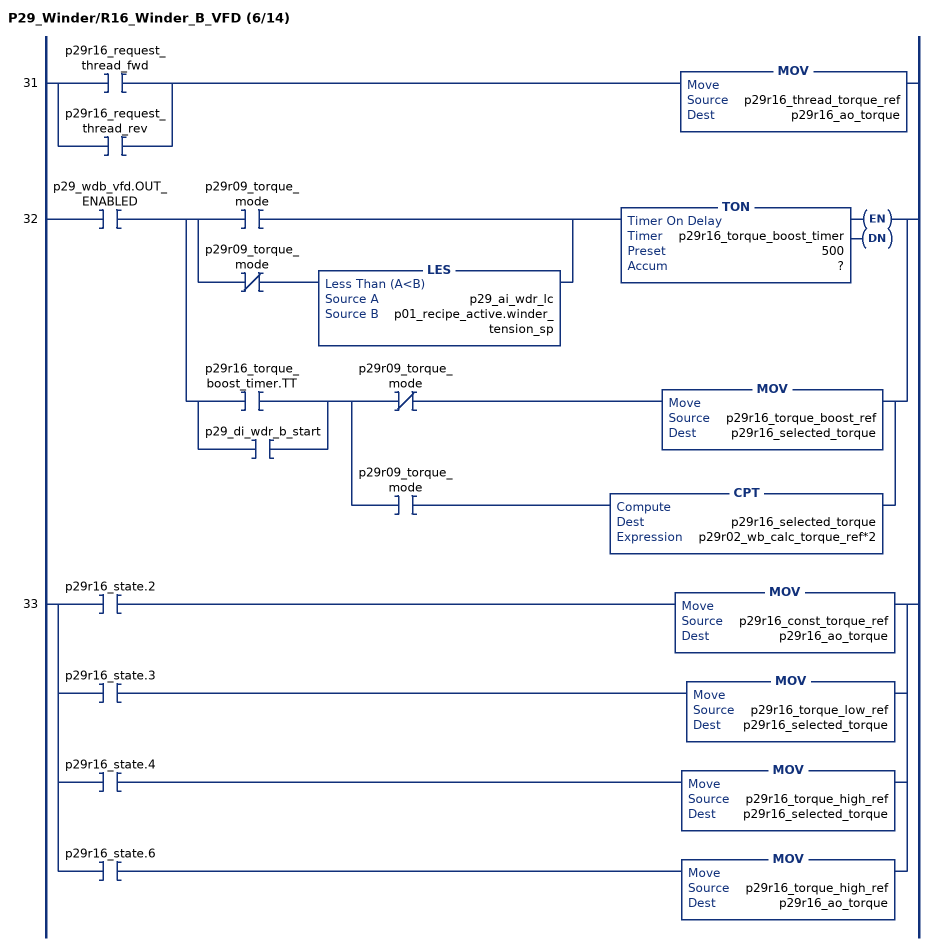
   31: [XIC(p29r16_request_thread_fwd) ,XIC(p29r16_request_thread_rev) ]MOV(p29r16_thread_torque_ref,p29r16_ao_torque);
   32: XIC(p29_wdb_vfd.OUT_ENABLED)[[XIC(p29r09_torque_mode) ,XIO(p29r09_torque_mode) LES(p29_ai_wdr_lc,p01_recipe_active.winder_tension_sp) ] TON(p29r16_torque_boost_timer,?,?) ,[XIC(p29r16_torque_boost_timer.TT) ,XIC(p29_di_wdr_b_start) ] [XIO(p29r09_torque_mode) MOV(p29r16_torque_boost_ref,p29r16_selected_torque) ,XIC(p29r09_torque_mode) CPT(p29r16_selected_torque,p29r02_wb_calc_torque_ref*2) ] ];
   33: [XIC(p29r16_state.2) MOV(p29r16_const_torque_ref,p29r16_ao_torque) ,XIC(p29r16_state.3) MOV(p29r16_torque_low_ref,p29r16_selected_torque) ,XIC(p29r16_state.4) MOV(p29r16_torque_high_ref,p29r16_selected_torque) ,XIC(p29r16_state.6) MOV(p29r16_torque_high_ref,p29r16_ao_torque) ];
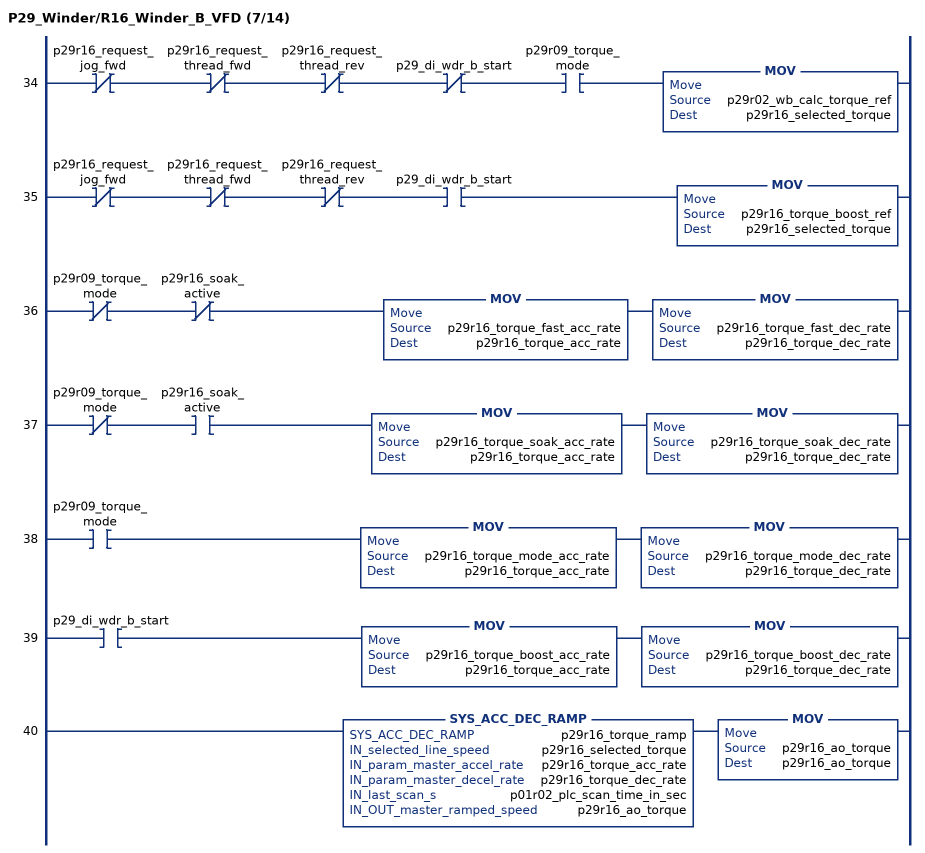
   34: XIO(p29r16_request_jog_fwd)XIO(p29r16_request_thread_fwd)XIO(p29r16_request_thread_rev)XIO(p29_di_wdr_b_start)XIC(p29r09_torque_mode)MOV(p29r02_wb_calc_torque_ref,p29r16_selected_torque);
   35: XIO(p29r16_request_jog_fwd)XIO(p29r16_request_thread_fwd)XIO(p29r16_request_thread_rev)XIC(p29_di_wdr_b_start)MOV(p29r16_torque_boost_ref,p29r16_selected_torque);
   36: XIO(p29r09_torque_mode)XIO(p29r16_soak_active)MOV(p29r16_torque_fast_acc_rate,p29r16_torque_acc_rate)MOV(p29r16_torque_fast_dec_rate,p29r16_torque_dec_rate);
   37: XIO(p29r09_torque_mode)XIC(p29r16_soak_active)MOV(p29r16_torque_soak_acc_rate,p29r16_torque_acc_rate)MOV(p29r16_torque_soak_dec_rate,p29r16_torque_dec_rate);
   38: XIC(p29r09_torque_mode)MOV(p29r16_torque_mode_acc_rate,p29r16_torque_acc_rate)MOV(p29r16_torque_mode_dec_rate,p29r16_torque_dec_rate);
   39: XIC(p29_di_wdr_b_start)MOV(p29r16_torque_boost_acc_rate,p29r16_torque_acc_rate)MOV(p29r16_torque_boost_dec_rate,p29r16_torque_dec_rate);
   40: SYS_ACC_DEC_RAMP(p29r16_torque_ramp,p29r16_selected_torque,p29r16_torque_acc_rate,p29r16_torque_dec_rate,p01r02_plc_scan_time_in_sec,p29r16_ao_torque)MOV(p29r16_ao_torque,p29r16_ao_torque);
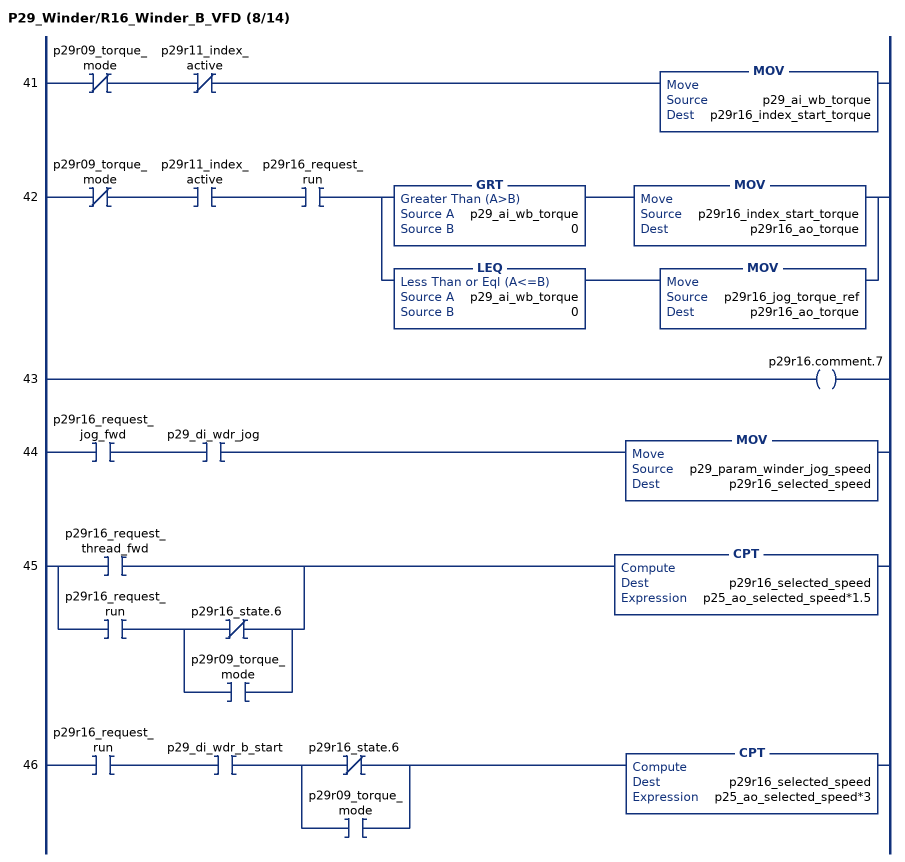
   41: XIO(p29r09_torque_mode)XIO(p29r11_index_active)MOV(p29_ai_wb_torque,p29r16_index_start_torque);
   42: XIO(p29r09_torque_mode)XIC(p29r11_index_active)XIC(p29r16_request_run)[GRT(p29_ai_wb_torque,0) MOV(p29r16_index_start_torque,p29r16_ao_torque) ,LEQ(p29_ai_wb_torque,0) MOV(p29r16_jog_torque_ref,p29r16_ao_torque) ];
   43: OTE(p29r16.comment.7);
   44: XIC(p29r16_request_jog_fwd)XIC(p29_di_wdr_jog)MOV(p29_param_winder_jog_speed,p29r16_selected_speed);
   45: [XIC(p29r16_request_thread_fwd) ,XIC(p29r16_request_run) [XIO(p29r16_state.6) ,XIC(p29r09_torque_mode) ] ]CPT(p29r16_selected_speed,p25_ao_selected_speed*1.5);
   46: XIC(p29r16_request_run)XIC(p29_di_wdr_b_start)[XIO(p29r16_state.6) ,XIC(p29r09_torque_mode) ]CPT(p29r16_selected_speed,p25_ao_selected_speed*3);
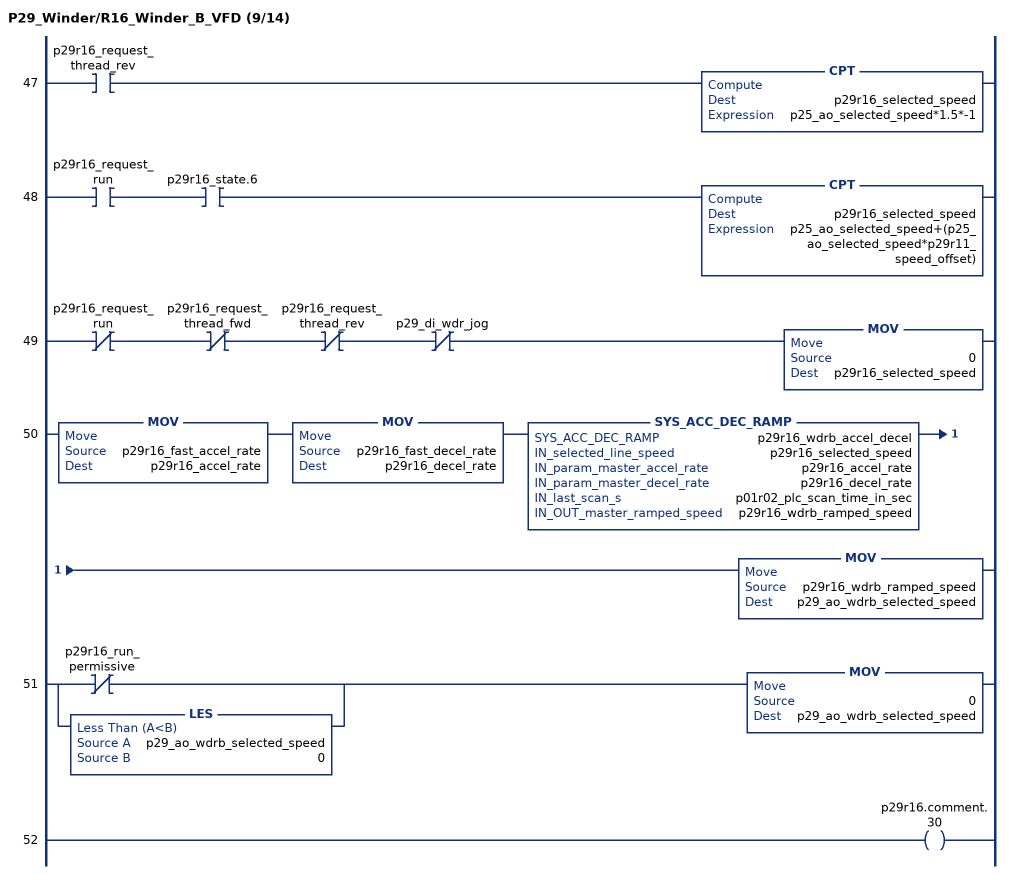
   47: XIC(p29r16_request_thread_rev)CPT(p29r16_selected_speed,p25_ao_selected_speed*1.5*-1);
   48: XIC(p29r16_request_run)XIC(p29r16_state.6)CPT(p29r16_selected_speed,p25_ao_selected_speed+(p25_ao_selected_speed*p29r11_speed_offset));
   49: XIO(p29r16_request_run)XIO(p29r16_request_thread_fwd)XIO(p29r16_request_thread_rev)XIO(p29_di_wdr_jog)MOV(0,p29r16_selected_speed);
   50: MOV(p29r16_fast_accel_rate,p29r16_accel_rate)MOV(p29r16_fast_decel_rate,p29r16_decel_rate)SYS_ACC_DEC_RAMP(p29r16_wdrb_accel_decel,p29r16_selected_speed,p29r16_accel_rate,p29r16_decel_rate,p01r02_plc_scan_time_in_sec,p29r16_wdrb_ramped_speed)MOV(p29r16_wdrb_ramped_speed,p29_ao_wdrb_selected_speed);
   51: [XIO(p29r16_run_permissive) ,LES(p29_ao_wdrb_selected_speed,0) ]MOV(0,p29_ao_wdrb_selected_speed);
   52: OTE(p29r16.comment.30);
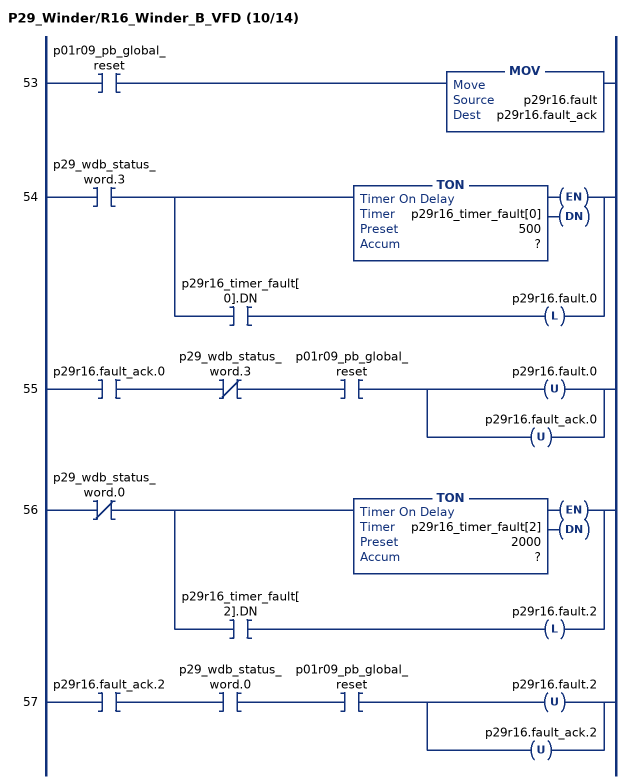
   53: XIC(p01r09_pb_global_reset)MOV(p29r16.fault,p29r16.fault_ack);
   54: XIC(p29_wdb_status_word.3)[TON(p29r16_timer_fault[0],?,?) ,XIC(p29r16_timer_fault[0].DN) OTL(p29r16.fault.0) ];
   55: XIC(p29r16.fault_ack.0)XIO(p29_wdb_status_word.3)XIC(p01r09_pb_global_reset)[OTU(p29r16.fault.0) ,OTU(p29r16.fault_ack.0) ];
   56: XIO(p29_wdb_status_word.0)[TON(p29r16_timer_fault[2],?,?) ,XIC(p29r16_timer_fault[2].DN) OTL(p29r16.fault.2) ];
   57: XIC(p29r16.fault_ack.2)XIC(p29_wdb_status_word.0)XIC(p01r09_pb_global_reset)[OTU(p29r16.fault.2) ,OTU(p29r16.fault_ack.2) ];
